// TIA Portal V17 export
// export: Created 2025-01-08T13:55:32.2808989Z, ExportSetting WithDefaults, DisplayName Totally Integrated Automation Portal, DisplayVersion V17, DisplayName TIA Portal Openness, DisplayVersion V17, DisplayName TIA Portal Version Control Interface, DisplayVersion V17, DisplayName SINAMICS Startdrive Advanced, DisplayVersion V17 Update2, DisplayName SINAMICS Startdrive G130, G150, S120, S150, SINAMICS MV, S210, DisplayVersion V17 Update2, DisplayName SINAMICS Startdrive G110M, G120, G120C, G120D, G120P, G115D, DisplayVersion V17 Update2, DisplayName STEP 7 Professional, DisplayVersion V17, DisplayName STEP 7 Safety, DisplayVersion V17, DisplayName WinCC Advanced, DisplayVersion V17
DATA_BLOCK "DB - 06_Errors_And_Warnings_HSM"   // DB98
{ S7_Optimized_Access := 'TRUE' }
VERSION : 0.1
// stored: AutoNumber false, DBAccessibleFromOPCUA true, DBAccessibleFromWebserver true, IsOnlyStoredInLoadMemory false, IsRetainMemResEnabled false, IsWriteProtectedInAS false, MemoryReserve 0
   VAR
      Alarm_1_HSM_NotReady_1 : Bool;
      Alarm_2_HSM_PLC_Conn_Faulty_1 : Bool;
      Alarm_3_HSM_NotReady_2 : Bool;
      Alarm_4_HSM_PLC_Conn_Faulty_2 : Bool;
      Alarm_5_HSM_NotReady_3 : Bool;
      Alarm_6_HSM_PLC_Conn_Faulty_3 : Bool;
      Alarm_7_Motor_Start_Error : Bool;
      Alarm_8_Motor_Position_Error : Bool;
      Alarm_9_Motor_Position_Control_Error : Bool;
      Alarm_10_Motor_Current_Target_Not_Reached : Bool;
      Alarm_11_Label_Gap_Not_Found : Bool;
      Alarm_12_Unwinder_Web_Break : Bool;
      Alarm_13_Web_End : Bool;
      Alarm_14_Motor_Overcurrent : Bool;
      Alarm_15_Dancer_Arm_Stop_Reached : Bool;
      Alarm_16 : Bool;
      Alarm_17_Rewinder_Web_Break : Bool;
      Alarm_18 : Bool;
      Alarm_19 : Bool;
      Alarm_20 : Bool;
      Warning_01_Find_Rotor_Position : Bool;
      Warning_02 : Bool;
      Warning_03_Number_Of_Labels_Reached : Bool;
      Warning_04_Low_Label_Reached : Bool;
      Warning_05_ZeroDownTime_Lan_Link_timeout : Bool;
      Warning_06_ZeroDownTime_Parameter_error : Bool;
      Warning_07 : Bool;
      Warning_08 : Bool;
      Warning_09_Roll_End_1 : Bool;
      Warning_10_Roll_End_2 : Bool;
      Warning_11_Roll_End_3 : Bool;
      Warning_10_HSM_1_PLC_DataTransmission_Error : Bool;
      Warning_13_HSM_2_PLC_DataTransmission_Error : Bool;
      Warning_14_HSM_3_PLC_DataTransmission_Error : Bool;
   END_VAR
BEGIN
END_DATA_BLOCK
